FUNCTION_BLOCK FB_Sercos_FSM_Test EXTENDS TcUnit.FB_TestSuite

TestStateS1();
TestStateS2();
TestStateS3();
TestStateS4();
TestStateS5a();
TestStateS5b();
TestStateS6();
TestStateS7();
TestStateS8();
TestEnableSequence();

METHOD PRIVATE GetEnableCommand : ST_Sercos_ControlWord
GetEnableCommand.b13_Halt := FALSE;
GetEnableCommand.b14_Enable := TRUE;
GetEnableCommand.b15_Start := TRUE;
END_METHOD

METHOD PRIVATE GetEnableHaltCommand : ST_Sercos_ControlWord
GetEnableHaltCommand.b13_Halt := TRUE;
GetEnableHaltCommand.b14_Enable := TRUE;
GetEnableHaltCommand.b15_Start := TRUE;
END_METHOD

METHOD PRIVATE GetErrorResetCommand : ST_Sercos_ControlWord
GetErrorResetCommand.b13_Halt := TRUE;
END_METHOD

METHOD PRIVATE GetHaltCommand : ST_Sercos_ControlWord
GetHaltCommand.b13_Halt := FALSE;
GetHaltCommand.b14_Enable := TRUE;
GetHaltCommand.b15_Start := TRUE;
END_METHOD

METHOD PRIVATE GetQuickStopCommand : ST_Sercos_ControlWord
GetQuickStopCommand.b14_Enable := TRUE;
GetQuickStopCommand.b15_Start := FALSE;
END_METHOD

METHOD PRIVATE GetRunCommand : ST_Sercos_ControlWord
GetRunCommand.b13_Halt := FALSE;
GetRunCommand.b14_Enable := TRUE;
GetRunCommand.b15_Start := TRUE;
END_METHOD

METHOD PRIVATE GetShutdownCommand : ST_Sercos_ControlWord
GetShutdownCommand.b14_Enable := FALSE;
END_METHOD

METHOD PRIVATE GetSwitchOnCommand : ST_Sercos_ControlWord
GetSwitchOnCommand.b14_Enable := TRUE;
END_METHOD

METHOD TestEnableSequence : BOOL
VAR
	fbSercosFSM 			: FB_Sercos_FSM;
	stExpectedStatus 		: ST_Sercos_StatusWord; 
	nMask 					: WORD;
	nResult 				: WORD;
	bResult 				: BOOL;
	nActualState			: INT;
	nExpectedState			: INT;
END_VAR
TEST('Enable S1');

nExpectedState := E_Sercos_State.S1_NotReadyToSwitchOn;
nActualState := fbSercosFSM.eState;

AssertEquals(Expected := nExpectedState,
             Actual := nActualState,
             Message := 'State is not correct');	 
TEST_FINISHED();

TEST('Enable S2');
fbSercosFSM();
nExpectedState := E_Sercos_State.S2_SwitchOnDisabled;
nActualState := fbSercosFSM.eState;

AssertEquals(Expected := nExpectedState,
             Actual := nActualState,
             Message := 'State is not correct');	 
TEST_FINISHED();

TEST('Enable S3');
fbSercosFSM.bPower := TRUE;
fbSercosFSM();
nExpectedState := E_Sercos_State.S3_ReadyToSwitchOn;
nActualState := fbSercosFSM.eState;

AssertEquals(Expected := nExpectedState,
             Actual := nActualState,
             Message := 'State is not correct');	 
TEST_FINISHED();

TEST('Enable S4');
fbSercosFSM.stControl := GetSwitchOnCommand();

fbSercosFSM();
nExpectedState := E_Sercos_State.S4_SwitchOn;
nActualState := fbSercosFSM.eState;

AssertEquals(Expected := nExpectedState,
             Actual := nActualState,
             Message := 'State is not correct');	 
TEST_FINISHED();

TEST('Enable S5a');
fbSercosFSM.stControl := GetEnableCommand();

fbSercosFSM();
nExpectedState := E_Sercos_State.S5a_DriveInOperation;
nActualState := fbSercosFSM.eState;

AssertEquals(Expected := nExpectedState,
             Actual := nActualState,
             Message := 'State is not correct');	 
TEST_FINISHED();
END_METHOD

METHOD TestStateS1 : BOOL
VAR
	fbSercosFSM 		: FB_Sercos_FSM;
	stExpectedStatus 	: ST_Sercos_StatusWord; 
	nMask 				: WORD;
	nResult 			: WORD;
	bResult 			: BOOL;
	nActualState		: INT;
	nExpectedState		: INT;
END_VAR
TEST('Set State S1');
fbSercosFSM.eState := E_Sercos_State.S1_NotReadyToSwitchOn;
fbSercosFSM();

stExpectedStatus.b15_ReadyToOperate 		:= FALSE;
stExpectedStatus.b14_ReadyToOperate 		:= FALSE;
stExpectedStatus.b13_Error 					:= FALSE;
stExpectedStatus.b7_QuickStop 				:= FALSE;
stExpectedStatus.b4_Halt 					:= FALSE;
stExpectedStatus.b3_CommandProcessing 		:= FALSE;

MEMCPY(ADR(nMask), ADR(stExpectedStatus), 2);
nResult := (2#1110000011011000 AND fbSercosFSM.nStatus);

AssertEquals(Expected := nMask,
             Actual := nResult,
             Message := 'Value is not correct');	 
TEST_FINISHED();

TEST('Transition S1>S2');
fbSercosFSM.eState := E_Sercos_State.S1_NotReadyToSwitchOn;
fbSercosFSM();

nExpectedState := E_Sercos_State.S2_SwitchOnDisabled;
nActualState := fbSercosFSM.eState;

AssertEquals(Expected := nExpectedState,
             Actual := nActualState,
             Message := 'State is not correct');	 
TEST_FINISHED();
END_METHOD

METHOD TestStateS2 : BOOL
VAR
	fbSercosFSM 		: FB_Sercos_FSM;
	stExpectedStatus 	: ST_Sercos_StatusWord; 
	nMask 				: WORD;
	nResult 			: WORD;
	bResult 			: BOOL;
	nActualState		: INT;
	nExpectedState		: INT;
END_VAR
TEST('Set State S2');
fbSercosFSM.eState := E_Sercos_State.S2_SwitchOnDisabled;
fbSercosFSM();

stExpectedStatus.b15_ReadyToOperate 		:= FALSE;
stExpectedStatus.b14_ReadyToOperate 		:= TRUE;
stExpectedStatus.b13_Error 					:= FALSE;
stExpectedStatus.b7_QuickStop 				:= FALSE;
stExpectedStatus.b4_Halt 					:= FALSE;
stExpectedStatus.b3_CommandProcessing 		:= FALSE;

MEMCPY(ADR(nMask), ADR(stExpectedStatus), 2);
nResult := (2#1110000011011000 AND fbSercosFSM.nStatus);

AssertEquals(Expected := nMask,
             Actual := nResult,
             Message := 'Value is not correct');	 
TEST_FINISHED();

TEST('Still State S2');
fbSercosFSM.bPower := FALSE;
fbSercosFSM.eState := E_Sercos_State.S2_SwitchOnDisabled;
fbSercosFSM();

nExpectedState := E_Sercos_State.S2_SwitchOnDisabled;
nActualState := fbSercosFSM.eState;

AssertEquals(Expected := nExpectedState,
             Actual := nActualState,
             Message := 'State is not correct');	 
TEST_FINISHED();

TEST('Transition S2>S3');
fbSercosFSM.bPower := TRUE;
fbSercosFSM.eState := E_Sercos_State.S2_SwitchOnDisabled;
fbSercosFSM();

nExpectedState := E_Sercos_State.S3_ReadyToSwitchOn;
nActualState := fbSercosFSM.eState;

AssertEquals(Expected := nExpectedState,
             Actual := nActualState,
             Message := 'State is not correct');	 
TEST_FINISHED();
END_METHOD

METHOD TestStateS3 : BOOL
VAR
	fbSercosFSM 		: FB_Sercos_FSM;
	stExpectedStatus 	: ST_Sercos_StatusWord; 
	nMask 				: WORD;
	nResult 			: WORD;
	bResult 			: BOOL;
	nActualState		: INT;
	nExpectedState		: INT;
END_VAR
TEST('Set State S3');
fbSercosFSM.eState := E_Sercos_State.S3_ReadyToSwitchOn;
fbSercosFSM();

stExpectedStatus.b15_ReadyToOperate 		:= TRUE;
stExpectedStatus.b14_ReadyToOperate 		:= FALSE;
stExpectedStatus.b13_Error 					:= FALSE;
stExpectedStatus.b7_QuickStop 				:= FALSE;
stExpectedStatus.b4_Halt 					:= FALSE;
stExpectedStatus.b3_CommandProcessing 		:= FALSE;

MEMCPY(ADR(nMask), ADR(stExpectedStatus), 2);
nResult := (2#1110000011011000 AND fbSercosFSM.nStatus);

AssertEquals(Expected := nMask,
             Actual := nResult,
             Message := 'Value is not correct');	 
TEST_FINISHED();

TEST('Transition S3>S2');
fbSercosFSM.bPower := FALSE;
fbSercosFSM.eState := E_Sercos_State.S3_ReadyToSwitchOn;
fbSercosFSM();

nExpectedState := E_Sercos_State.S2_SwitchOnDisabled;
nActualState := fbSercosFSM.eState;

AssertEquals(Expected := nExpectedState,
             Actual := nActualState,
             Message := 'State is not correct');	 
TEST_FINISHED();

TEST('Transition S3>S7');
fbSercosFSM.bPower := TRUE;
fbSercosFSM.bError := TRUE;
fbSercosFSM.eState := E_Sercos_State.S3_ReadyToSwitchOn;
fbSercosFSM();

nExpectedState := E_Sercos_State.S7_FaultReactionActive;
nActualState := fbSercosFSM.eState;

AssertEquals(Expected := nExpectedState,
             Actual := nActualState,
             Message := 'State is not correct');	 
TEST_FINISHED();

TEST('Transition S3>S4');
fbSercosFSM.bError := FALSE;
fbSercosFSM.stControl := GetSwitchOnCommand();
fbSercosFSM.eState := E_Sercos_State.S3_ReadyToSwitchOn;
fbSercosFSM();

nExpectedState := E_Sercos_State.S4_SwitchOn;
nActualState := fbSercosFSM.eState;

AssertEquals(Expected := nExpectedState,
             Actual := nActualState,
             Message := 'State is not correct');	 
TEST_FINISHED();
END_METHOD

METHOD TestStateS4 : BOOL
VAR
	fbSercosFSM 		: FB_Sercos_FSM;
	stExpectedStatus 	: ST_Sercos_StatusWord; 
	nMask 				: WORD;
	nResult 			: WORD;
	bResult 			: BOOL;
	nActualState		: INT;
	nExpectedState		: INT;
END_VAR
TEST('Set State S4');
fbSercosFSM.eState := E_Sercos_State.S4_SwitchOn;
fbSercosFSM();

stExpectedStatus.b15_ReadyToOperate 		:= TRUE;
stExpectedStatus.b14_ReadyToOperate 		:= TRUE;
stExpectedStatus.b13_Error 					:= FALSE;
stExpectedStatus.b7_QuickStop 				:= FALSE;
stExpectedStatus.b4_Halt 					:= FALSE;
stExpectedStatus.b3_CommandProcessing 		:= FALSE;

MEMCPY(ADR(nMask), ADR(stExpectedStatus), 2);
nResult := (2#1110000011011000 AND fbSercosFSM.nStatus);

AssertEquals(Expected := nMask,
             Actual := nResult,
             Message := 'Value is not correct');	 
TEST_FINISHED();

TEST('Transition S4>S2');
fbSercosFSM.bPower := FALSE;
fbSercosFSM.eState := E_Sercos_State.S4_SwitchOn;
fbSercosFSM();
fbSercosFSM();

nExpectedState := E_Sercos_State.S2_SwitchOnDisabled;
nActualState := fbSercosFSM.eState;

AssertEquals(Expected := nExpectedState,
             Actual := nActualState,
             Message := 'State is not correct');	 
TEST_FINISHED();

TEST('Transition S4>S3');
fbSercosFSM.bPower := TRUE;
fbSercosFSM.eState := E_Sercos_State.S4_SwitchOn;
fbSercosFSM.stControl := GetShutdownCommand();
fbSercosFSM();

nExpectedState := E_Sercos_State.S3_ReadyToSwitchOn;
nActualState := fbSercosFSM.eState;

AssertEquals(Expected := nExpectedState,
             Actual := nActualState,
             Message := 'State is not correct');	 
TEST_FINISHED();

TEST('Transition S4>S7');
fbSercosFSM.bPower := TRUE;
fbSercosFSM.bError := TRUE;
fbSercosFSM.eState := E_Sercos_State.S4_SwitchOn;
fbSercosFSM();

nExpectedState := E_Sercos_State.S7_FaultReactionActive;
nActualState := fbSercosFSM.eState;

AssertEquals(Expected := nExpectedState,
             Actual := nActualState,
             Message := 'State is not correct');	 
TEST_FINISHED();

TEST('Transition S4>S5b');
fbSercosFSM.bError := FALSE;
fbSercosFSM.stControl := GetEnableHaltCommand();
fbSercosFSM.eState := E_Sercos_State.S4_SwitchOn;
fbSercosFSM();

nExpectedState := E_Sercos_State.S5b_Halt;
nActualState := fbSercosFSM.eState;

AssertEquals(Expected := nExpectedState,
             Actual := nActualState,
             Message := 'State is not correct');	 
TEST_FINISHED();

TEST('Transition S4>S5a');
fbSercosFSM.bError := FALSE;
fbSercosFSM.stControl := GetEnableCommand();
fbSercosFSM.eState := E_Sercos_State.S4_SwitchOn;
fbSercosFSM();

nExpectedState := E_Sercos_State.S5a_DriveInOperation;
nActualState := fbSercosFSM.eState;

AssertEquals(Expected := nExpectedState,
             Actual := nActualState,
             Message := 'State is not correct');	 
TEST_FINISHED();
END_METHOD

METHOD TestStateS5a : BOOL
VAR
	fbSercosFSM 		: FB_Sercos_FSM;
	stExpectedStatus 	: ST_Sercos_StatusWord; 
	nMask 				: WORD;
	nResult 			: WORD;
	bResult 			: BOOL;
	nActualState		: INT;
	nExpectedState		: INT;
END_VAR
TEST('Set State S5a');
fbSercosFSM.eState := E_Sercos_State.S5a_DriveInOperation;
fbSercosFSM();

stExpectedStatus.b15_ReadyToOperate 		:= TRUE;
stExpectedStatus.b14_ReadyToOperate 		:= TRUE;
stExpectedStatus.b13_Error 					:= FALSE;
stExpectedStatus.b7_QuickStop 				:= FALSE;
stExpectedStatus.b4_Halt 					:= FALSE;
stExpectedStatus.b3_CommandProcessing 		:= TRUE;

MEMCPY(ADR(nMask), ADR(stExpectedStatus), 2);
nResult := (2#1110000011011000 AND fbSercosFSM.nStatus);

AssertEquals(Expected := nMask,
             Actual := nResult,
             Message := 'Value is not correct');	 
TEST_FINISHED();

TEST('Transition S5a>S2');
fbSercosFSM.bPower := FALSE;
fbSercosFSM.eState := E_Sercos_State.S5a_DriveInOperation;
fbSercosFSM();
fbSercosFSM();

nExpectedState := E_Sercos_State.S2_SwitchOnDisabled;
nActualState := fbSercosFSM.eState;

AssertEquals(Expected := nExpectedState,
             Actual := nActualState,
             Message := 'State is not correct');	 
TEST_FINISHED();

TEST('Transition S5a>S7');
fbSercosFSM.bPower := TRUE;
fbSercosFSM.bError := TRUE;
fbSercosFSM.eState := E_Sercos_State.S5a_DriveInOperation;
fbSercosFSM();

nExpectedState := E_Sercos_State.S7_FaultReactionActive;
nActualState := fbSercosFSM.eState;

AssertEquals(Expected := nExpectedState,
             Actual := nActualState,
             Message := 'State is not correct');	 
TEST_FINISHED();

TEST('Transition S5a>S3');
fbSercosFSM.bError := FALSE;
fbSercosFSM.bPower := TRUE;
fbSercosFSM.eState := E_Sercos_State.S5a_DriveInOperation;
fbSercosFSM.stControl := GetShutdownCommand();
fbSercosFSM();

nExpectedState := E_Sercos_State.S3_ReadyToSwitchOn;
nActualState := fbSercosFSM.eState;

AssertEquals(Expected := nExpectedState,
             Actual := nActualState,
             Message := 'State is not correct');	 
TEST_FINISHED();

TEST('Transition S5a>S6');
fbSercosFSM.bError := FALSE;
fbSercosFSM.bPower := TRUE;
fbSercosFSM.eState := E_Sercos_State.S5a_DriveInOperation;
fbSercosFSM.stControl := GetQuickStopCommand();
fbSercosFSM();

nExpectedState := E_Sercos_State.S6_QuickStop;
nActualState := fbSercosFSM.eState;

AssertEquals(Expected := nExpectedState,
             Actual := nActualState,
             Message := 'State is not correct');	 
TEST_FINISHED();

TEST('Transition S5a>S5b');
fbSercosFSM.bError := FALSE;
fbSercosFSM.bPower := TRUE;
fbSercosFSM.stControl := GetEnableHaltCommand();
fbSercosFSM.eState := E_Sercos_State.S5a_DriveInOperation;
fbSercosFSM();

nExpectedState := E_Sercos_State.S5b_Halt;
nActualState := fbSercosFSM.eState;

AssertEquals(Expected := nExpectedState,
             Actual := nActualState,
             Message := 'State is not correct');	 
TEST_FINISHED();
END_METHOD

METHOD TestStateS5b : BOOL
VAR
	fbSercosFSM 		: FB_Sercos_FSM;
	stExpectedStatus 	: ST_Sercos_StatusWord; 
	nMask 				: WORD;
	nResult 			: WORD;
	bResult 			: BOOL;
	nActualState		: INT;
	nExpectedState		: INT;
END_VAR
TEST('Set State S5b');
fbSercosFSM.eState := E_Sercos_State.S5b_Halt;
fbSercosFSM();

stExpectedStatus.b15_ReadyToOperate 		:= TRUE;
stExpectedStatus.b14_ReadyToOperate 		:= TRUE;
stExpectedStatus.b13_Error 					:= FALSE;
stExpectedStatus.b7_QuickStop 				:= FALSE;
stExpectedStatus.b4_Halt 					:= TRUE;
stExpectedStatus.b3_CommandProcessing 		:= FALSE;

MEMCPY(ADR(nMask), ADR(stExpectedStatus), 2);
nResult := (2#1110000011011000 AND fbSercosFSM.nStatus);

AssertEquals(Expected := nMask,
             Actual := nResult,
             Message := 'Value is not correct');	 
TEST_FINISHED();

TEST('Transition S5b>S2');
fbSercosFSM.bPower := FALSE;
fbSercosFSM.eState := E_Sercos_State.S5b_Halt;
fbSercosFSM();

nExpectedState := E_Sercos_State.S2_SwitchOnDisabled;
nActualState := fbSercosFSM.eState;

AssertEquals(Expected := nExpectedState,
             Actual := nActualState,
             Message := 'State is not correct');	 
TEST_FINISHED();

TEST('Transition S5b>S7');
fbSercosFSM.bPower := TRUE;
fbSercosFSM.bError := TRUE;
fbSercosFSM.eState := E_Sercos_State.S5b_Halt;
fbSercosFSM();

nExpectedState := E_Sercos_State.S7_FaultReactionActive;
nActualState := fbSercosFSM.eState;

AssertEquals(Expected := nExpectedState,
             Actual := nActualState,
             Message := 'State is not correct');	 
TEST_FINISHED();

TEST('Transition S5b>S3');
fbSercosFSM.bError := FALSE;
fbSercosFSM.bPower := TRUE;
fbSercosFSM.eState := E_Sercos_State.S5b_Halt;
fbSercosFSM.stControl := GetShutdownCommand();
fbSercosFSM();

nExpectedState := E_Sercos_State.S3_ReadyToSwitchOn;
nActualState := fbSercosFSM.eState;

AssertEquals(Expected := nExpectedState,
             Actual := nActualState,
             Message := 'State is not correct');	 
TEST_FINISHED();

TEST('Transition S5b>S6');
fbSercosFSM.bError := FALSE;
fbSercosFSM.bPower := TRUE;
fbSercosFSM.eState := E_Sercos_State.S5b_Halt;
fbSercosFSM.stControl := GetQuickStopCommand();
fbSercosFSM();

nExpectedState := E_Sercos_State.S6_QuickStop;
nActualState := fbSercosFSM.eState;

AssertEquals(Expected := nExpectedState,
             Actual := nActualState,
             Message := 'State is not correct');	 
TEST_FINISHED();

TEST('Transition S5b>S5a');
fbSercosFSM.bError := FALSE;
fbSercosFSM.bPower := TRUE;
fbSercosFSM.stControl := GetEnableCommand();
fbSercosFSM.eState := E_Sercos_State.S5b_Halt;
fbSercosFSM();

nExpectedState := E_Sercos_State.S5a_DriveInOperation;
nActualState := fbSercosFSM.eState;

AssertEquals(Expected := nExpectedState,
             Actual := nActualState,
             Message := 'State is not correct');	 
TEST_FINISHED();
END_METHOD

METHOD TestStateS6 : BOOL
VAR
	fbSercosFSM 		: FB_Sercos_FSM;
	stExpectedStatus 	: ST_Sercos_StatusWord; 
	nMask 				: WORD;
	nResult 			: WORD;
	bResult 			: BOOL;
	nActualState		: INT;
	nExpectedState		: INT;
END_VAR
TEST('Set State S6');
fbSercosFSM.eState := E_Sercos_State.S6_QuickStop;
fbSercosFSM();

stExpectedStatus.b15_ReadyToOperate 		:= TRUE;
stExpectedStatus.b14_ReadyToOperate 		:= TRUE;
stExpectedStatus.b13_Error 					:= FALSE;
stExpectedStatus.b7_QuickStop 				:= TRUE;
stExpectedStatus.b4_Halt 					:= TRUE;
stExpectedStatus.b3_CommandProcessing 		:= FALSE;

MEMCPY(ADR(nMask), ADR(stExpectedStatus), 2);
nResult := (2#1110000011011000 AND fbSercosFSM.nStatus);

AssertEquals(Expected := nMask,
             Actual := nResult,
             Message := 'Value is not correct');	 
TEST_FINISHED();

TEST('Transition S6>S2');
fbSercosFSM.bPower := FALSE;
fbSercosFSM.eState := E_Sercos_State.S6_QuickStop;
fbSercosFSM();
fbSercosFSM();

nExpectedState := E_Sercos_State.S2_SwitchOnDisabled;
nActualState := fbSercosFSM.eState;

AssertEquals(Expected := nExpectedState,
             Actual := nActualState,
             Message := 'State is not correct');	 
TEST_FINISHED();

TEST('Transition S6>S3');
fbSercosFSM.bPower := TRUE;
fbSercosFSM.eState := E_Sercos_State.S6_QuickStop;
fbSercosFSM.stControl := GetShutdownCommand();
fbSercosFSM();

nExpectedState := E_Sercos_State.S3_ReadyToSwitchOn;
nActualState := fbSercosFSM.eState;

AssertEquals(Expected := nExpectedState,
             Actual := nActualState,
             Message := 'State is not correct');	 
TEST_FINISHED();

TEST('Transition S6>S7');
fbSercosFSM.bPower := TRUE;
fbSercosFSM.bError := TRUE;
fbSercosFSM.eState := E_Sercos_State.S6_QuickStop;
fbSercosFSM();

nExpectedState := E_Sercos_State.S7_FaultReactionActive;
nActualState := fbSercosFSM.eState;

AssertEquals(Expected := nExpectedState,
             Actual := nActualState,
             Message := 'State is not correct');	 
TEST_FINISHED();

TEST('Transition S6>S5b');
fbSercosFSM.bError := FALSE;
fbSercosFSM.stControl := GetEnableHaltCommand();
fbSercosFSM.eState := E_Sercos_State.S6_QuickStop;
fbSercosFSM();

nExpectedState := E_Sercos_State.S5b_Halt;
nActualState := fbSercosFSM.eState;

AssertEquals(Expected := nExpectedState,
             Actual := nActualState,
             Message := 'State is not correct');	 
TEST_FINISHED();

TEST('Transition S6>S5a');
fbSercosFSM.bError := FALSE;
fbSercosFSM.stControl := GetEnableCommand();
fbSercosFSM.eState := E_Sercos_State.S6_QuickStop;
fbSercosFSM();

nExpectedState := E_Sercos_State.S5a_DriveInOperation;
nActualState := fbSercosFSM.eState;

AssertEquals(Expected := nExpectedState,
             Actual := nActualState,
             Message := 'State is not correct');	 
TEST_FINISHED();
END_METHOD

METHOD TestStateS7 : BOOL
VAR
	fbSercosFSM 		: FB_Sercos_FSM;
	stExpectedStatus 	: ST_Sercos_StatusWord; 
	nMask 				: WORD;
	nResult 			: WORD;
	bResult 			: BOOL;
	nActualState		: INT;
	nExpectedState		: INT;
END_VAR
TEST('Set State S7');
fbSercosFSM.eState := E_Sercos_State.S7_FaultReactionActive;
fbSercosFSM();

stExpectedStatus.b15_ReadyToOperate 		:= TRUE;
stExpectedStatus.b14_ReadyToOperate 		:= TRUE;
stExpectedStatus.b13_Error 					:= TRUE;
stExpectedStatus.b7_QuickStop 				:= FALSE;
stExpectedStatus.b4_Halt 					:= FALSE;
stExpectedStatus.b3_CommandProcessing 		:= FALSE;

MEMCPY(ADR(nMask), ADR(stExpectedStatus), 2);
nResult := (2#1110000011011000 AND fbSercosFSM.nStatus);

AssertEquals(Expected := nMask,
             Actual := nResult,
             Message := 'Value is not correct');	 
TEST_FINISHED();

TEST('Transition S7>S2');
fbSercosFSM.bPower := FALSE;
fbSercosFSM.eState := E_Sercos_State.S7_FaultReactionActive;
fbSercosFSM();

nExpectedState := E_Sercos_State.S2_SwitchOnDisabled;
nActualState := fbSercosFSM.eState;

AssertEquals(Expected := nExpectedState,
             Actual := nActualState,
             Message := 'State is not correct');	 
TEST_FINISHED();

TEST('Transition S7>S8');
fbSercosFSM.bPower := TRUE;
fbSercosFSM.eState := E_Sercos_State.S7_FaultReactionActive;
fbSercosFSM();

nExpectedState := E_Sercos_State.S8_Fault;
nActualState := fbSercosFSM.eState;

AssertEquals(Expected := nExpectedState,
             Actual := nActualState,
             Message := 'State is not correct');	 
TEST_FINISHED();
END_METHOD

METHOD TestStateS8 : BOOL
VAR
	fbSercosFSM 		: FB_Sercos_FSM;
	stExpectedStatus 	: ST_Sercos_StatusWord; 
	nMask 				: WORD;
	nResult 			: WORD;
	bResult 			: BOOL;
	nActualState		: INT;
	nExpectedState		: INT;
END_VAR
TEST('Set State S8');
fbSercosFSM.eState := E_Sercos_State.S8_Fault;
fbSercosFSM();

stExpectedStatus.b15_ReadyToOperate 		:= TRUE;
stExpectedStatus.b14_ReadyToOperate 		:= FALSE;
stExpectedStatus.b13_Error 					:= TRUE;
stExpectedStatus.b7_QuickStop 				:= FALSE;
stExpectedStatus.b4_Halt 					:= FALSE;
stExpectedStatus.b3_CommandProcessing 		:= FALSE;

MEMCPY(ADR(nMask), ADR(stExpectedStatus), 2);
nResult := (2#1110000011011000 AND fbSercosFSM.nStatus);

AssertEquals(Expected := nMask,
             Actual := nResult,
             Message := 'Value is not correct');	 
TEST_FINISHED();

TEST('Transition S8>S2');
fbSercosFSM.bPower := FALSE;
fbSercosFSM.eState := E_Sercos_State.S8_Fault;
fbSercosFSM.stControl := GetErrorResetCommand();
fbSercosFSM();

nExpectedState := E_Sercos_State.S2_SwitchOnDisabled;
nActualState := fbSercosFSM.eState;

AssertEquals(Expected := nExpectedState,
             Actual := nActualState,
             Message := 'State is not correct');	 
TEST_FINISHED();
END_METHOD

END_FUNCTION_BLOCK

(* stored: Version 1.1.0.1, ProductVersion 3.1.4024.12
   POU FB_Sercos_FSM_Test: Id {e2d93bb2-8db7-065e-0371-9c388aae7b6c}, SpecialFunc None
   Method GetEnableCommand: Id {5de932be-52cc-0f39-05bc-ec07a41466a5}
   Method GetEnableHaltCommand: Id {3de8d8af-49a1-05b6-2ffb-18e21b0d70b7}
   Method GetErrorResetCommand: Id {3a9661e4-58ec-091e-1035-d08ad5253a8b}
   Method GetHaltCommand: Id {e0e1aba9-b928-06bb-13ea-1ba116a1a445}
   Method GetQuickStopCommand: Id {e766e34a-9dd7-00a8-2e9e-48997c85dedf}
   Method GetRunCommand: Id {08dcdec4-46cf-05d9-0d20-322cd750613e}
   Method GetShutdownCommand: Id {f5d673d5-ac1d-096c-216f-9ec726cbde62}
   Method GetSwitchOnCommand: Id {03275183-f8ee-06c5-3e42-61c0ee012bd6}
   Method TestEnableSequence: Id {d8c371ba-e014-0996-1a03-d3a15eb80fd8}
   Method TestStateS1: Id {3bc78463-bff2-0672-2100-2c0792a00ca4}
   Method TestStateS2: Id {84a637f2-5728-08bf-2613-c5e1569edc81}
   Method TestStateS3: Id {8d0b5a15-c593-09ec-00e8-18ae6f2ad90d}
   Method TestStateS4: Id {5cf18472-704a-0647-2a38-a4b08f399007}
   Method TestStateS5a: Id {741205e9-622a-0fc8-2a85-021e628e757c}
   Method TestStateS5b: Id {4ec04249-868d-0ea0-07fc-71985e93ffae}
   Method TestStateS6: Id {57b40535-3ec2-0d01-1f67-a5fa7f5a1498}
   Method TestStateS7: Id {99db4e42-849b-0bcb-271e-052486b3270e}
   Method TestStateS8: Id {2e830f06-f3cd-0c0d-26f0-f946e1d46979} *)
